{attribute 'GeneratedUsingTerminal: EP3351-2022-0016'}
{attribute addProperty BoxType "EP3351-2022-0016"}
{attribute addProperty Id "EtcSlaveTerminalBaseAIBridge_InputsAT %I*AIBridge_Inputs_555AA1E89AISupply_InputsAT %I*AISupply_Inputs_555AA1E89WcStateAT %I*WcState_9091E0EB2InfoDataAT %I*InfoData_32EB74EA10"}
{attribute addProperty CRC "371360226"}
{attribute addProperty Size "30"}
TYPE EP3351_162281E2 EXTENDS EtcSlaveTerminalBase :
STRUCT
	{attribute addProperty Name "AIBridge_Inputs"}
	AIBridge_Inputs : AIBridge_Inputs_555AA1E8;
	{attribute addProperty Name "AISupply_Inputs"}
	AISupply_Inputs : AISupply_Inputs_555AA1E8;
	{attribute addProperty Name "WcState"}
	WcState : WcState_9091E0EB;
	{attribute addProperty Name "InfoData"}
	InfoData : InfoData_32EB74EA;
END_STRUCT
END_TYPE

(* stored: Version 1.2.0.0, ProductVersion 3.1.4024.9
   DUT EP3351_162281E2: Id {26d2b40f-c694-4517-aed0-2d86193208e6} *)
